PROGRAM MAIN
VAR
	runonce:BOOL:=FALSE;
END_VAR

IF NOT runonce THEN
	ADSLOGSTR( msgCtrlMask := ADSLOG_MSGTYPE_ERROR OR ADSLOG_MSGTYPE_LOG, msgFmtStr := 'PLC Msg', strArg := '');
	runonce:=TRUE;
END_IF

END_PROGRAM

(* stored: Version 1.1.0.1, ProductVersion 3.1.4024.13
   POU MAIN: Id {af6a45e9-1729-44e9-9f23-c238a8c97ac0}, SpecialFunc None *)
